SYSTEM CounterNetwork
  (* Version 1.0, 2022-06-20, AK115394 *)
  APPLICATION CounterNetworkApp
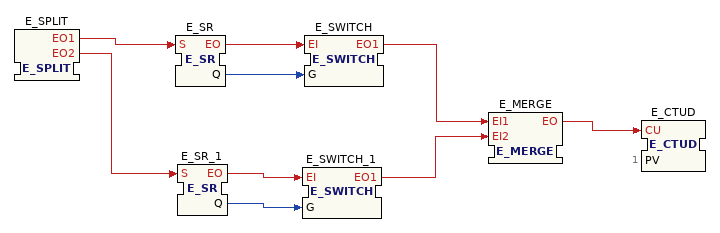
    FBS
      E_SR : E_SR;
      E_SWITCH : E_SWITCH;
      E_SPLIT : E_SPLIT;
      E_SR_1 : E_SR;
      E_SWITCH_1 : E_SWITCH;
      E_MERGE : E_MERGE;
      E_CTUD : E_CTUD(PV := 1);
    END_FBS
    EVENT_CONNECTIONS
      E_SPLIT.EO1 TO E_SR.S;
      E_SR.EO TO E_SWITCH.EI;
      E_SPLIT.EO2 TO E_SR_1.S;
      E_SR_1.EO TO E_SWITCH_1.EI;
      E_SWITCH.EO1 TO E_MERGE.EI1;
      E_SWITCH_1.EO1 TO E_MERGE.EI2;
      E_MERGE.EO TO E_CTUD.CU;
    END_CONNECTIONS
    DATA_CONNECTIONS
      E_SR.Q TO E_SWITCH.G;
      E_SR_1.Q TO E_SWITCH_1.G;
    END_CONNECTIONS
  END_APPLICATION
END_SYSTEM
